# B&R Automation Studio project FASTorySystems (part 6)

#### Types.typ - Exported data types
```iecst
TYPE
	fdMove6DParametersType : 	STRUCT
		Position : fdMove6DParPositionType;
		Limits : fdMove6DParLimitsType;
		Velocity : fdMove6DParVelocityType;
		Mode : McAcp6DMoveModeEnum;
	END_STRUCT;
	fdMove6DParPositionType : 	STRUCT
		X : REAL;
		Y : REAL;
		Z : REAL;
		Rx : REAL;
		Ry : REAL;
		Rz : REAL;
	END_STRUCT;
	fdMove6DParLimitsType : 	STRUCT
		Velocity_InPlane : REAL;
		Velocity_Rx : REAL;
		Velocity_Ry : REAL;
		Velocity_Rz : REAL;
		Velocity_Z : REAL;
		Acceleration : REAL;
	END_STRUCT;
	fdMove6DParVelocityType : 	STRUCT
		InPlane : REAL;
		Z : REAL;
		Rx : REAL;
		Ry : REAL;
		Rz : REAL;
	END_STRUCT;
END_TYPE
```

#### Constants.var - Exported constants
```iecst
VAR CONSTANT
	fdMAX_STATION_SHUTTLE_COUNT : DINT := 4;
END_VAR
```

#### FastLib.fun - Exported functions and function blocks
```iecst
FUNCTION_BLOCK fdStationQueueControl
	VAR_INPUT
		Enable : {REDUND_UNREPLICABLE} BOOL;
		ReleaseShuttles : {REDUND_UNREPLICABLE} BOOL;
		SelectNextShuttle : {REDUND_UNREPLICABLE} BOOL;
		ShuttleList : {REDUND_UNREPLICABLE} ARRAY[0..fdMAX_STATION_SHUTTLE_COUNT] OF MpTrafficShuttleInfoType;
		ShuttleCapacity : {REDUND_UNREPLICABLE} DINT; (*Count how many shuttles process station can handle*)
		pStationControl : REFERENCE TO MpTrafficStationControl;
	END_VAR
	VAR_OUTPUT
		ShuttleReleaseDone : BOOL;
		ShuttleReleaseError : BOOL;
		ReleaseShuttle : BOOL;
		LastReleasedShuttleID : UINT;
	END_VAR
	VAR
		state : DINT;
		i : DINT;
		index : DINT;
		shuttleID : UINT;
		lastSelectedIndex : UINT;
	END_VAR
END_FUNCTION_BLOCK

FUNCTION_BLOCK fdTiltAround
	VAR_INPUT
		Execute : {REDUND_UNREPLICABLE} BOOL;
		MaxAngle : {REDUND_UNREPLICABLE} REAL;
		Steps : {REDUND_UNREPLICABLE} DINT;
		Velocity : McAcp6DShortAxAxesType;
		Shuttle : REFERENCE TO Mc6DShuttleType;
	END_VAR
	VAR_OUTPUT
		Acknowledge : BOOL;
		Error : BOOL;
	END_VAR
	VAR
		state : DINT;
		step : DINT;
		MoveShortAxis : MC_BR_MoveShortAxis_Acp6D;
	END_VAR
END_FUNCTION_BLOCK

FUNCTION_BLOCK fdWaitUntilAllDone
	VAR_INPUT
		Execute : {REDUND_UNREPLICABLE} BOOL;
		Shuttles : {REDUND_UNREPLICABLE} ARRAY[0..fdMAX_STATION_SHUTTLE_COUNT] OF Mc6DShuttleType;
	END_VAR
	VAR_OUTPUT
		Done : BOOL;
		Error : BOOL;
		WaitingFor : UINT;
	END_VAR
	VAR
		state : DINT;
		i : DINT;
		ShGetInfo : MC_BR_ShGetInfo_Acp6D;
	END_VAR
END_FUNCTION_BLOCK

FUNCTION_BLOCK fdPulse
	VAR_INPUT
		Execute : {REDUND_UNREPLICABLE} BOOL;
		T_on : {REDUND_UNREPLICABLE} TIME;
		T_off : {REDUND_UNREPLICABLE} TIME;
	END_VAR
	VAR_OUTPUT
		Q : BOOL;
	END_VAR
	VAR
		state : DINT;
		TON_on : TON;
		TON_off : TON;
	END_VAR
END_FUNCTION_BLOCK

FUNCTION_BLOCK fdLampSequence
	VAR_INPUT
		Execute : {REDUND_UNREPLICABLE} BOOL;
	END_VAR
	VAR_OUTPUT
		Lamp1 : BOOL;
		Lamp2 : BOOL;
		Lamp3 : BOOL;
	END_VAR
	VAR
		state : DINT;
		TON_delay : TON;
	END_VAR
END_FUNCTION_BLOCK

FUNCTION_BLOCK fdFindZone
	VAR_INPUT
		Assembly : REFERENCE TO Mc6DAssemblyType; (*The assembly reference establishes the connection between the function block and the assembly.*)
		Execute : BOOL;
		Name : STRING[32];
	END_VAR
	VAR_OUTPUT
		ZoneFound : BOOL;
		ZoneNotFound : BOOL;
		Error : BOOL;
		Zone : Mc6DZoneType; (* Zone reference *)
		ZoneInfo : McAcp6DGetZoneAddInfoType;
	END_VAR
	VAR
		state : DINT;
		i : DINT;
		AsmGetZone : MC_BR_AsmGetZone_Acp6D;
		lastZoneID : UINT;
	END_VAR
END_FUNCTION_BLOCK

FUNCTION_BLOCK fdMove6D
	VAR_INPUT
		Shuttle : REFERENCE TO Mc6DShuttleType; (*The assembly reference establishes the connection between the function block and the assembly.*)
		Execute : BOOL;
		Parameters : fdMove6DParametersType;
	END_VAR
	VAR_OUTPUT
		Acknowledge : BOOL;
		Done : BOOL;
		Error : BOOL;
	END_VAR
	VAR
		state : DINT;
		i : DINT;
		ShGetInfo : MC_BR_ShGetInfo_Acp6D;
		Move6D : MC_BR_Move6D_Acp6D;
	END_VAR
END_FUNCTION_BLOCK
```

#### fdReleaseQueuingShuttle.st
```iecst
(*  *)
FUNCTION_BLOCK fdStationQueueControl

	IF NOT Enable THEN
		state := 0;
		ReleaseShuttle := FALSE;
		SelectNextShuttle := FALSE;
		LastReleasedShuttleID := 0;
		ShuttleReleaseDone := FALSE;
		ShuttleReleaseError := FALSE;
		RETURN;
	END_IF;

	CASE state OF
		0:
			// -----------------------------------------------------------------
			SelectNextShuttle := FALSE;

			IF ReleaseShuttles THEN
				state := 20;
			ELSIF pStationControl.Info.NumOccupyingShuttles > ShuttleCapacity THEN
				// Station is executing current process and there is no room for more shuttles ->
				// release queuing extra shuttles straight forward
				state := 10;
			END_IF;
		10:
			// Check if we have our last arrived shuttle selected
			// -----------------------------------------------------------------
			IF pStationControl.SelectedShuttle.ShuttleID = pStationControl.Info.LastArrivedShuttle.ShuttleID THEN
	  			state := 12;
			ELSE
				lastSelectedIndex := pStationControl.SelectedShuttle.Index;
				SelectNextShuttle := FALSE;
				state := 11;
			END_IF;
		11:
			// Select next shuttle in the queue
			// -----------------------------------------------------------------
			SelectNextShuttle := TRUE;
			// Wait until selection changes
			IF lastSelectedIndex <> pStationControl.SelectedShuttle.Index THEN
				SelectNextShuttle := FALSE;
				state := 10;
			END_IF;
		12:
			// Release the queuing shuttle
			// -----------------------------------------------------------------
			ReleaseShuttle := TRUE;

			IF pStationControl.ReleaseDone THEN
				LastReleasedShuttleID := pStationControl.SelectedShuttle.ShuttleID;
				ReleaseShuttle := FALSE;
				state := 0;
			ELSIF pStationControl.ReleaseAborted THEN
				LastReleasedShuttleID := 0;
				ReleaseShuttle := FALSE;
				state := 0;
			END_IF;

		20:
			// Initialize for realease
			// -----------------------------------------------------------------
			i := 0;
			state := 21;
		21:
			// Select the next requested shuttle from the shuttle list
			// -----------------------------------------------------------------
			shuttleID := 0;

			WHILE i <= fdMAX_STATION_SHUTTLE_COUNT DO
				IF ShuttleList[i].ShuttleID > 0 THEN
					shuttleID := ShuttleList[i].ShuttleID;
					i := i + 1;
					EXIT;
				END_IF;
				i := i + 1;
			END_WHILE;

			IF shuttleID > 0 THEN
				// Found shuttle to release
				state := 22;
			ELSE
				// No more shuttles to release
	  			state := 100;
			END_IF;
		22:
			// Check if we have our last arrived shuttle selected
			// -----------------------------------------------------------------
			IF pStationControl.SelectedShuttle.ShuttleID = shuttleID THEN
				state := 24;
			ELSE
				lastSelectedIndex := pStationControl.SelectedShuttle.Index;
				SelectNextShuttle := FALSE;
				state := 23;
			END_IF;
		23:
			// Select next shuttle in the queue
			// -----------------------------------------------------------------
			SelectNextShuttle := TRUE;
			// Wait until selection changes
			IF lastSelectedIndex <> pStationControl.SelectedShuttle.Index THEN
				SelectNextShuttle := FALSE;
				i := 0;
				state := 21;
			END_IF;
		24:
			// Release the queuing shuttle
			// -----------------------------------------------------------------
			ReleaseShuttle := TRUE;

			IF pStationControl.ReleaseDone THEN
				LastReleasedShuttleID := pStationControl.SelectedShuttle.ShuttleID;
				ReleaseShuttle := FALSE;
				state := 21;
			ELSIF pStationControl.ReleaseAborted THEN
				LastReleasedShuttleID := 0;
				ReleaseShuttle := FALSE;
				state := 21;
			END_IF;

//
//		22:
//			// Find shuttle from stations shuttle table
//			// -----------------------------------------------------------------
//			state := 21; // Assume we dont find shuttle and just return straight to next one
//
//			FOR index := 0 TO pStationControl.Info.NumOccupyingShuttles DO
//				IF pStationControl.SelectedShuttle.ShuttleID = shuttleID THEN
//					state := 23;
//					EXIT;
//				END_IF
//				pStationControl(SelectNextShuttle := TRUE);
//				pStationControl(SelectNextShuttle := FALSE);
//			END_FOR;
//
//		23:
//			// Release the waiting shuttle
//			// -----------------------------------------------------------------
//			ReleaseShuttle := TRUE;
//
//			IF pStationControl.ReleaseDone THEN
//				ReleaseShuttle := FALSE;
//				state := 21;
//			END_IF;
		100:
			// Done
			// -----------------------------------------------------------------
			IF NOT ReleaseShuttles THEN
				state := 0;
			END_IF;
		200:
			// Error
			// -----------------------------------------------------------------
			IF NOT ReleaseShuttles THEN
				state := 0;
			END_IF;
	END_CASE;

	ShuttleReleaseDone := (state = 100);
	ShuttleReleaseError := (state = 200);

END_FUNCTION_BLOCK
```

#### fdTiltAround.st
```iecst
(*  *)
FUNCTION_BLOCK fdTiltAround

	IF NOT Execute THEN
		MoveShortAxis.Execute := FALSE;
		step := 0;
		state := 0;
	END_IF;

	CASE state OF
		0:
			IF Execute THEN
				state := 10;
			END_IF;
		10:
			IF step > Steps THEN
				state := 100;
			ELSE
				MoveShortAxis.Parameters.Position.Rx := MaxAngle * SIN((2 * brmPI / Steps) * step);
				MoveShortAxis.Parameters.Position.Ry := MaxAngle * COS((2 * brmPI / Steps) * step);
				MoveShortAxis.Parameters.Position.Rz := 0;
				MoveShortAxis.Parameters.Position.Z := 0.004;
				state := 20;
			END_IF;
		20:
			MoveShortAxis.Execute := TRUE;

			IF MoveShortAxis.Acknowledge THEN
				MoveShortAxis.Execute := FALSE;
				step := step + 1;
				state := 10;
			END_IF;
		100:
//			MoveShortAxis.Parameters.Position.Rx := 0;
//			MoveShortAxis.Parameters.Position.Ry := 0;
//			MoveShortAxis.Parameters.Position.Rz := 0;
//			MoveShortAxis.Parameters.Position.Z := 0.001;
//			MoveShortAxis.Execute := TRUE;
//
//			IF MoveShortAxis.Done OR MoveShortAxis.Acknowledge THEN
//				MoveShortAxis.Execute := FALSE;
//				step := step + 1;
//				state := 101;
//			END_IF;

			IF NOT Execute THEN
				state := 0;
			END_IF;
	END_CASE;

	MoveShortAxis.Shuttle := ADR(Shuttle);
	MoveShortAxis.Parameters.Mode :=  mcACP6D_MOVE_ABSOLUTE;
	MoveShortAxis.Parameters.Velocity := Velocity;
	MoveShortAxis();

	Acknowledge := (state = 100);
	Error := MoveShortAxis.Error;

END_FUNCTION_BLOCK
```

#### fdWaitUntilIdle.st
```iecst
(*  *)
FUNCTION_BLOCK fdWaitUntilAllDone

	IF NOT Execute THEN
		state := 0;
		i := 0;
		ShGetInfo.Execute := FALSE;
		WaitingFor := 0;
	END_IF;

	CASE state OF
		0:
			IF Execute THEN
				state := 10;
			END_IF;
		10:
			IF i > fdMAX_STATION_SHUTTLE_COUNT THEN
				state := 100;
			ELSE
				IF Shuttles[i].controlif = 0 THEN
					// Not a valid shuttle reference. Move to next item in the list
					i := i + 1;
				ELSE
					state := 20;
				END_IF;
			END_IF;
		20:
			ShGetInfo.Execute := TRUE;

			IF ShGetInfo.Done THEN
				WaitingFor := ShGetInfo.ShuttleInfo.ShuttleID;

				IF (ShGetInfo.ShuttleInfo.State =  mcACP6D_SH_STATE_IDLING) AND (ShGetInfo.ShuttleInfo.MotionBuffer.NumberOfCommands = 0) THEN
					i := i + 1;
					state := 10;
				END_IF;
				ShGetInfo.Execute := FALSE;

			ELSIF ShGetInfo.Error THEN
				ShGetInfo.Execute := FALSE;
				state := 101;
			END_IF;
		100:
			IF NOT Execute THEN
				state := 0;
			END_IF;
	END_CASE;

	ShGetInfo.Shuttle := ADR(Shuttles[i]);
	ShGetInfo();

	Done := (state = 100);
	Error := ShGetInfo.Error;

END_FUNCTION_BLOCK
```

#### fdPulse.st
```iecst
(*  *)
FUNCTION_BLOCK fdPulse

	IF NOT Execute THEN
		state := 0;
	END_IF;

	CASE state OF
		0:
			IF Execute THEN
				state := 10;
			END_IF;
		10:
			IF TON_on.Q THEN
	  			state := 20;
			END_IF;
		20:
			IF TON_off.Q THEN
				state := 10;
			END_IF;
		100:
			IF NOT Execute THEN
				state := 0;
			END_IF;
	END_CASE;

	TON_on.IN := (state = 10);
	TON_on.PT := T_on;
	TON_on();

	TON_off.IN := (state = 20);
	TON_off.PT := T_off;
	TON_off();

	Q := (state = 10);

END_FUNCTION_BLOCK
```

#### fdLampSequence.st
```iecst
(*  *)
FUNCTION_BLOCK fdLampSequence

	IF NOT Execute THEN
		state := 0;
	END_IF;

	CASE state OF
		0:
			IF Execute THEN
				state := 10;
			END_IF;
		10:
			TON_delay.IN := TRUE;
			IF TON_delay.Q THEN
				TON_delay.IN := FALSE;
	  			state := 20;
			END_IF;
		20:
			TON_delay.IN := TRUE;
			IF TON_delay.Q THEN
				TON_delay.IN := FALSE;
				state := 30;
			END_IF;
		30:
			TON_delay.IN := TRUE;
			IF TON_delay.Q THEN
				TON_delay.IN := FALSE;
				state := 10;
			END_IF;
	END_CASE;

	TON_delay.PT := T#150ms;
	TON_delay();

	Lamp1 := (state = 10);
	Lamp2 := (state = 20);
	Lamp3 := (state = 30);

END_FUNCTION_BLOCK
```

#### fdFindZone.st
```iecst
(*  *)
FUNCTION_BLOCK fdFindZone

	IF NOT Execute THEN
		state := 0;
		i := 0;
		AsmGetZone.Enable := FALSE;
		ZoneFound := FALSE;
		ZoneNotFound := FALSE;
		Error := FALSE;
		brsmemset(ADR(ZoneInfo), 0, SIZEOF(ZoneInfo));
		brsmemset(ADR(Zone), 0, SIZEOF(Zone));
	END_IF;

	CASE state OF
		0:
			// --------------------------------------------
			IF Execute THEN
				state := 10;
			END_IF;
		10:
			// --------------------------------------------
			AsmGetZone.Enable := TRUE;
			IF AsmGetZone.Valid THEN
				IF AsmGetZone.TotalCount = 0 THEN
					state := 101;
				ELSE
					state := 20;
				END_IF;
			END_IF;
		20:
			// --------------------------------------------
			lastZoneID := AsmGetZone.AdditionalInfo.ZoneID;

			IF brsmemcmp(ADR(AsmGetZone.AdditionalInfo.Name), ADR(Name), SIZEOF(Name)) = 0 THEN
				// Names match -> found
				Zone := AsmGetZone.Zone;
				ZoneInfo := AsmGetZone.AdditionalInfo;
				state := 100;
			ELSE
				IF AsmGetZone.RemainingCount = 0 THEN
					state := 101;
				ELSE
					state := 30;
				END_IF;
			END_IF;
		30:
			// --------------------------------------------
			IF AsmGetZone.AdditionalInfo.ZoneID <> lastZoneID THEN
				state := 20;
			END_IF;

		100:
			// --------------------------------------------
			ZoneFound := TRUE;
		101:
			// --------------------------------------------
			ZoneNotFound := TRUE;
		102:
			// --------------------------------------------
			Error := TRUE;
	END_CASE;

	AsmGetZone.Assembly := ADR(Assembly);
	AsmGetZone.Next := (state = 30);
	AsmGetZone();

END_FUNCTION_BLOCK
```

#### fdMove6D.st
```iecst
(*  *)
FUNCTION_BLOCK fdMove6D

//	IF NOT Execute THEN
//		state := 0;
//		i := 0;
//	END_IF;
//
//	CASE state OF
//		0:
//			// --------------------------------------------
//			IF Execute THEN
//				state := 10;
//			END_IF;
//		100:
//			// --------------------------------------------
//			ZoneFound := TRUE;
//		101:
//			// --------------------------------------------
//			ZoneNotFound := TRUE;
//		102:
//			// --------------------------------------------
//			Error := TRUE;
//	END_CASE;
//
//	Move6D.Assembly := ADR(Shuttle);
//	AsmGetZone.Next := (state = 30);
//	AsmGetZone();
//
//	ShGetInfo.Shuttle := ADR(Shuttle);
//	ShGetInfo();

END_FUNCTION_BLOCK
```

### global.var
```iecst
VAR
	gFastDemo : FastDemoType := (0);
END_VAR
```

### global.typ
```iecst
(*
Program: FastDemo

Description
(short summary)

*)
(*========== INPUTS ==========*)

TYPE
	FastDemoInputCommandType : 	STRUCT
		Activate : BOOL;
	END_STRUCT;
	FastDemoInputStatusType : 	STRUCT
		SetupComplete : BOOL;
	END_STRUCT;
	FastDemoInputType : 	STRUCT
		Force : BOOL;
		Command : FastDemoInputCommandType;
		Status : FastDemoInputStatusType;
	END_STRUCT;
END_TYPE

(*========== OUTPUTS ==========*)

TYPE
	FastDemoOutputCommandType : 	STRUCT
		NewCommand : BOOL;
	END_STRUCT;
	FastDemoOutputStatusType : 	STRUCT
		NewStatus : BOOL;
	END_STRUCT;
	FastDemoOutputType : 	STRUCT
		Command : FastDemoOutputCommandType;
		Status : FastDemoOutputStatusType;
	END_STRUCT;
END_TYPE

(*========== ERRORS ==========*)
(*========== SETTINGS ==========*)

TYPE
	FastDemoSettingsType : 	STRUCT
		Enable : BOOL;
	END_STRUCT;
END_TYPE

(*========== INTERFACE ==========*)

TYPE
	FastDemoType : 	STRUCT
		Error : GeneralErrorInfoType;
		Input : FastDemoInputType;
		Output : FastDemoOutputType;
		Settings : FastDemoSettingsType;
	END_STRUCT;
END_TYPE
```

### Program Logical/src/FastDemo/FastDemo (IEC)

#### FastDemo.st
```iecst
PROGRAM _INIT

    // Access the task interface
    task ACCESS ADR(gFastDemo);

    // Register module config interface for common setup/parametrization functionality
    //fb.MpRecipeRegPar_settings(MpLink := ADR(gSystemSettings), Enable := TRUE , PVName := ADR('gFastDemo.settings'), Category := ADR('FastDemo'));

    // Check for simulator
    //task.IsSimulated := DiagCpuIsSimulated();

    // PackML setup
    // =================================================================================================================
    em.Setup.Name := 'FastDemo';
	em.Setup.ParentName := 'Main';

END_PROGRAM

PROGRAM _CYCLIC

    // Access task interface
    // =================================================================================================================
    task ACCESS ADR(gFastDemo);

    // Inputs
    // =================================================================================================================
    IF NOT task.Input.Force THEN

    END_IF

	// Task state machine
	// =================================================================================================================
	// PackML state machine execution
	PackML_state_machine;

	// Detect state change events
	// =================================================================================================================
	// Record information which state caused abort
	fb.R_TRIG_Abort(CLK := em.Command.Abort);

	IF fb.R_TRIG_Abort.Q THEN
		task.Error.State := em.StateCurrent;
		task.Error.SubState := em.SubState;
		task.Error.Description := em.StateInfo;
	END_IF;

	// State change event
	fb.rtStateComplete(CLK := em.Command.StateComplete);

	IF fb.rtStateComplete.Q THEN
		em.StateInfo := '';
		brsmemset(ADR(actions_state), 0, SIZEOF(actions_state));

		// Record information which state caused abort
		IF em.StateCurrent = STATE_ABORTING THEN
			task.Error.State := local.lastState;
			task.Error.SubState := local.lastSubState;
			task.Error.Description := local.lastStateInfo;
		END_IF;

		FOR station_num := 0 TO STATION_COUNT DO
			// Reset station commands when major state changes
			stations[station_num].State := 0;
			brsmemset(ADR(stations[station_num].Var), 0, SIZEOF(stations[station_num].Var));
			brsmemset(ADR(stations[station_num].Commands), 0, SIZEOF(stations[station_num].Commands));
			stations[station_num].Macro.Execute := FALSE;
		END_FOR;
	END_IF;

	// Substate changed event
	IF em.SubState <> local.lastSubState THEN
		em.StateInfo := '';
		brsmemset(ADR(actions_substate), 0, SIZEOF(actions_substate));
		local.lastSubState := em.SubState;
	END_IF;

	// PackML equipment module
	// =================================================================================================================
	em();

	// Function calls
    // =================================================================================================================
	fb.TrafficControl.Enable := TRUE;
	fb.TrafficControl.MpLink := ADR(TrafficManager_x6d_1);
	fb.TrafficControl.ActivateRecipe := actions_substate.traffic_activate_recipe;
	fb.TrafficControl.DeactivateRecipe := actions_substate.traffic_deactivate_recipe;
	fb.TrafficControl.ErrorReset := actions_state.error_reset;
	fb.TrafficControl.Halt := actions_substate.traffic_halt;
	fb.TrafficControl.Recover := actions_substate.traffic_recover;
	fb.TrafficControl.Resume := actions_substate.traffic_resume;
	fb.TrafficControl.Stop := actions_substate.traffic_stop;
	fb.TrafficControl();

	fb.TON_RecoverTimeout.IN := fb.TrafficControl.RecoverBuffered;
	fb.TON_RecoverTimeout.PT := T#5s;
	fb.TON_RecoverTimeout();

	fb.TrafficMonitor.Enable := TRUE;
	fb.TrafficMonitor.MpLink := ADR(TrafficManager_x6d_1);
	fb.TrafficMonitor();

	fb.MacroDelete.Assembly := ADR(gAssembly6D_Big);
	fb.MacroDelete.Execute := actions_substate.macro_delete;
	fb.MacroDelete.Command := mcACP6D_MACRO_DELETE_ALL;
	fb.MacroDelete();

	fb.GroupGet.Assembly := ADR(gAssembly6D_Big);
	fb.GroupGet.Enable := actions_state.group_get_enable;
	fb.GroupGet();

	fb.GroupDelete.Execute := actions_substate.group_delete;
	fb.GroupDelete();

	// Perform all common station operations
	FOR station_num := 0 TO STATION_COUNT DO
		station ACCESS ADR(stations[station_num]);

		// Station control
		station.Control.MpLink := ADR(TrafficManager_x6d_1);
		station.Control.ErrorReset := actions_state.error_reset;
		station.Control.Release := station.Operation.StationQueueControl.ReleaseShuttle;
		station.Control.SelectNextShuttle := station.Operation.StationQueueControl.SelectNextShuttle;
		station.Control();

		station.Operation.StationQueueControl.Enable := actions_state.activate_queue_control;
		station.Operation.StationQueueControl.ReleaseShuttles := station.Commands.Release;
		station.Operation.StationQueueControl.pStationControl := ADR(station.Control);
		station.Operation.StationQueueControl();

		// Movement
		station.Operation.MoveInPlane.Execute := station.Commands.MoveInPlane;
		station.Operation.MoveInPlane();

		station.Operation.MoveArc.Execute := station.Commands.MoveArc;
		station.Operation.MoveArc();

		station.Operation.Move6D.Execute := station.Commands.Move6D;
		station.Operation.Move6D();

		station.Operation.MoveShortAxis.Execute := station.Commands.MoveShortAxis;
		station.Operation.MoveShortAxis();

		station.Operation.Spin.Execute := station.Commands.Spin;
		station.Operation.Spin();

		station.Operation.TiltAround.Execute := station.Commands.TiltAround;
		station.Operation.TiltAround();

		station.Operation.SunPlanet.Execute := station.Commands.ChangePlanet;
		station.Operation.SunPlanet();

		station.Operation.GetShuttleInfo.Execute := station.Commands.GetShuttleInfo;
		station.Operation.GetShuttleInfo();

		// Macro
		station.Macro.MacroCreate.Assembly := ADR(gAssembly6D_Big);
		station.Macro.MacroCreate.Parameters.Name := station.Macro.Name;
		station.Macro.MacroCreate.Execute := station.Commands.Macro.Create;
		station.Macro.MacroCreate();

		station.Macro.MacroSave.Shuttle := ADR(station.Macro.Shuttle);
		station.Macro.MacroSave.Execute := station.Commands.Macro.Save;
		station.Macro.MacroSave();

		station.Macro.MacroRun.Name := station.Macro.Name;
		station.Macro.MacroRun.Execute := station.Macro.Execute;
		station.Macro.MacroRun();

		// Group
		station.Group.GroupCreate.Execute := station.Commands.Group.Create;
		station.Group.GroupCreate.Assembly := ADR(gAssembly6D_Big);
		station.Group.GroupCreate();

		station.Group.GroupClear.Execute := station.Commands.Group.Clear;
		station.Group.GroupClear.ShuttleGroup := ADR(station.Group.ShuttleGroup);
		station.Group.GroupClear();

		station.Group.GroupAddShuttle.Execute := station.Commands.Group.AddShuttle;
		station.Group.GroupAddShuttle.ShuttleGroup := ADR(station.Group.ShuttleGroup);
		station.Group.GroupAddShuttle();

		station.Group.GroupCoupleCtrl.Execute := station.Commands.Group.ChangeCoupling;
		station.Group.GroupCoupleCtrl.ShuttleGroup := ADR(station.Group.ShuttleGroup);
		station.Group.GroupCoupleCtrl();

		// Zone
		station.Zone.ZoneCreate.Execute := station.Commands.Zone.Create;
		station.Zone.ZoneCreate.Assembly := ADR(gAssembly6D_Big);
		station.Zone.ZoneCreate();

		station.Zone.ZoneGetBarrierInfo.Execute := station.Commands.Zone.GetBarrierInfo;
		station.Zone.ZoneGetBarrierInfo.Zone := ADR(station.Zone.Zone);
		station.Zone.ZoneGetBarrierInfo();

		station.Zone.FindZone.Execute := station.Commands.Zone.Find;
		station.Zone.FindZone.Assembly := ADR(gAssembly6D_Big);
		station.Zone.FindZone();

		// Virtual
		station.Virtual.VirtualShCreate.Execute := station.Commands.CreateVirtualShuttle;
		station.Virtual.VirtualShCreate.Assembly := ADR(gAssembly6D_Big);
		station.Virtual.VirtualShCreate();

		// Wait
		station.Operation.WaitCommandLabel.Execute := station.Commands.WaitCommandLabel;
		station.Operation.WaitCommandLabel();

		station.Operation.WaitUntilAllDone.Execute := station.Commands.WaitUntilAllDone;
		station.Operation.WaitUntilAllDone();
	END_FOR;

	// Task outputs
	// =================================================================================================================

	// Task diagnostics
	// =================================================================================================================
	gTasks.FastDemo.State := em.StateCurrent;
	gTasks.FastDemo.SubState := em.SubState;
	gTasks.FastDemo.Mode := em.ModeID;
	gTasks.FastDemo.StateComplete := em.Command.StateComplete;
	gTasks.FastDemo.StateInfo := em.StateInfo;
	gTasks.FastDemo.WaitingForTask := em.Info.WaitingFor.Name;
	gTasks.FastDemo.Error := task.Error;

END_PROGRAM

PROGRAM _EXIT

END_PROGRAM
```

#### local.typ
```iecst
TYPE
	FastDemoFbType : 	STRUCT
		MpRecipeRegPar_settings : BOOL;
		TrafficControl : MpTrafficControl;
		TrafficMonitor : MpTrafficMonitor;
		rtStateComplete : R_TRIG;
		MacroDelete : MC_BR_MacroDelete_Acp6D;
		GroupGet : MC_BR_AsmGetShGroup_Acp6D;
		GroupDelete : MC_BR_ShGroupDelete_Acp6D;
		R_TRIG_Abort : R_TRIG;
		TON_RecoverTimeout : TON;
	END_STRUCT;
	FastDemoLocalType : 	STRUCT
		lastState : DINT;
		lastSubState : DINT;
		lastStateInfo : STRING[80];
		allGroupsDeleted : BOOL;
	END_STRUCT;
	FastDemoActionsStateType : 	STRUCT
		error_reset : BOOL;
		group_get_enable : BOOL;
		activate_queue_control : BOOL;
	END_STRUCT;
	FastDemoActionsSubstateType : 	STRUCT
		traffic_activate_recipe : BOOL; (*Task actions are not automatically reset*)
		traffic_deactivate_recipe : BOOL; (*Task actions are not automatically reset*)
		traffic_halt : BOOL;
		traffic_recover : BOOL;
		traffic_resume : BOOL;
		traffic_stop : BOOL;
		macro_delete : BOOL;
		group_delete : BOOL;
	END_STRUCT;
	FastDemoHmiType : 	STRUCT
		isRunning : BOOL;
	END_STRUCT;
END_TYPE

(**)
(*Stations*)

TYPE
	FastDemoStationType : 	STRUCT
		State : DINT;
		SequenceStep : DINT;
		Shuttles : ARRAY[0..STATION_SHUTTLE_LAST_INDEX]OF MpTrafficShuttleInfoType;
		ShuttleCount : DINT;
		Var : FastDemoStationVarType;
		Control : MpTrafficStationControl;
		Commands : FastDemoStationCommandsType;
		Operation : FastDemoStationOperationType;
		Macro : FastDemoStationMacroType;
		Group : FastDemoStationGroupType;
		Zone : FastDemoStationZoneType;
		Virtual : FastDemoStationVirtualType;
	END_STRUCT;
	FastDemoStationVarType : 	STRUCT
		PreviousState : DINT;
		StateInfo : STRING[80];
		LoopNum : DINT;
	END_STRUCT;
	FastDemoStationCommandsType : 	STRUCT
		Release : BOOL;
		Macro : FastDemoStationMacroCommandsType;
		Group : FastDemoStationGroupCommandsType;
		Zone : FastDemoStationZoneCommandsType;
		CreateVirtualShuttle : BOOL;
		MoveInPlane : BOOL;
		MoveArc : BOOL;
		MoveShortAxis : BOOL;
		Move6D : BOOL;
		Spin : BOOL;
		TiltAround : BOOL;
		ChangePlanet : BOOL;
		WaitCommandLabel : BOOL;
		GetShuttleInfo : BOOL;
		WaitUntilAllDone : BOOL;
	END_STRUCT;
	FastDemoStationMacroCommandsType : 	STRUCT
		Create : BOOL;
		Save : BOOL;
		Delete : BOOL;
	END_STRUCT;
	FastDemoStationGroupCommandsType : 	STRUCT
		Create : BOOL;
		Clear : BOOL;
		Delete : BOOL;
		AddShuttle : BOOL;
		ChangeCoupling : BOOL;
	END_STRUCT;
	FastDemoStationZoneCommandsType : 	STRUCT
		Create : BOOL;
		Find : BOOL;
		GetBarrierInfo : BOOL;
	END_STRUCT;
	FastDemoStationOperationType : 	STRUCT
		StationQueueControl : fdStationQueueControl;
		MoveInPlane : MC_BR_MoveInPlane_Acp6D;
		MoveArc : MC_BR_MoveArc_Acp6D;
		Spin : MC_BR_RotaryMotionSpin_Acp6D;
		Move6D : MC_BR_Move6D_Acp6D;
		MoveShortAxis : MC_BR_MoveShortAxis_Acp6D;
		TiltAround : fdTiltAround;
		SunPlanet : MC_BR_ShPlanet_Acp6D;
		WaitCommandLabel : MC_BR_ShWaitCmdLb_Acp6D;
		GetShuttleInfo : MC_BR_ShGetInfo_Acp6D;
		WaitUntilAllDone : fdWaitUntilAllDone;
	END_STRUCT;
	FastDemoStationMacroType : 	STRUCT
		Shuttle : Mc6DShuttleType;
		Name : STRING[32];
		Execute : BOOL;
		MacroCreate : MC_BR_MacroCreate_Acp6D;
		MacroSave : MC_BR_MacroSave_Acp6D;
		MacroRun : MC_BR_MacroRun_Acp6D;
	END_STRUCT;
	FastDemoStationGroupType : 	STRUCT
		ShuttleGroup : Mc6DShuttleGroupType;
		GroupCreate : MC_BR_ShGroupCreate_Acp6D;
		GroupClear : MC_BR_ShGroupClear_Acp6D;
		GroupCoupleCtrl : MC_BR_ShGroupCoupleCtrl_Acp6D;
		GroupAddShuttle : MC_BR_ShGroupAddShuttle_Acp6D;
	END_STRUCT;
	FastDemoStationZoneType : 	STRUCT
		Zone : Mc6DZoneType;
		Name : STRING[32];
		ZoneCreate : MC_BR_ZoneCreate_Acp6D;
		ZoneGetBarrierInfo : MC_BR_ZoneGetBarrierInfo_Acp6D;
		FindZone : fdFindZone;
	END_STRUCT;
	FastDemoStationVirtualType : 	STRUCT
		Shuttle : Mc6DShuttleType;
		ShuttleID : UINT;
		VirtualShCreate : MC_BR_VirtualShCreate_Acp6D;
	END_STRUCT;
END_TYPE
```

#### local.var
```iecst
VAR
	task : REFERENCE TO FastDemoType;
	local : FastDemoLocalType;
	fb : FastDemoFbType;
	hmi : FastDemoHmiType;
	actions_state : FastDemoActionsStateType;
	actions_substate : FastDemoActionsSubstateType;
END_VAR
(* ----- PackML ----- *)
VAR
	em : EquipmentModule;
END_VAR
(*----- Stations ----*)
VAR
	station_num : {REDUND_UNREPLICABLE} DINT := 0;
	str : STRING[80];
	i : DINT;
END_VAR
VAR CONSTANT
	STATION_COUNT : DINT := 7;
	STATION_SHUTTLE_COUNT : DINT := 4;
	STATION_SHUTTLE_LAST_INDEX : DINT := STATION_SHUTTLE_COUNT-1;
END_VAR
VAR
	stations : ARRAY[0..STATION_COUNT] OF FastDemoStationType;
	station : REFERENCE TO FastDemoStationType;
END_VAR
```

#### PackML.st
```iecst
// PackML state machine. Split into different sections that handle
// different logical sequences of PackML stadards' steps
// INFO: Add mode specific code into states by adding CASE structure
// 	CASE em.ModeID OF
//		MODE_PRODUCTION:
//			*CODE*;
//		MODE_MAINTENANCE:
//			*CODE*;
//		MODE_MANUAL:
//			*CODE*;
//		END_CASE
// -----------------------------------------------------------------

ACTION PackML_state_machine:
	// =================================================================================================================
    // Global PackML events
    // =================================================================================================================

    // =================================================================================================================
    // Normal work sequence
    // =================================================================================================================
    CASE em.StateCurrent OF
        STATE_STOPPED:
            em.StateInfo := '';
            // -----------------------------------------------------------------
            em.Command.StateComplete := TRUE;

        STATE_RESETTING:
			CASE em.SubState OF
				0:
					em.StateInfo := 'Reset traffic control errors';
					// -----------------------------------------------------------------
					actions_state.error_reset := TRUE;
					IF NOT fb.TrafficControl.Error THEN
	  					em.SubState := 10;
					END_IF;
				10:
					em.StateInfo := 'Delete all macros';
					// -----------------------------------------------------------------
					actions_substate.macro_delete := TRUE;
					IF fb.MacroDelete.Done THEN
						FOR station_num := 0 TO STATION_COUNT DO
							brsmemset(ADR(stations[station_num].Macro.Shuttle), 0, SIZEOF(stations[station_num].Macro.Shuttle));
						END_FOR;
						em.SubState := 20;
					END_IF;
				20:
					em.StateInfo := 'Delete all groups';
					// -----------------------------------------------------------------
					actions_state.group_get_enable := TRUE;

					IF fb.GroupGet.Valid THEN
						IF fb.GroupGet.TotalCount = 0 THEN
							// Clear all shuttle group references
							FOR station_num := 0 TO STATION_COUNT DO
	  							brsmemset(ADR(stations[station_num].Group.ShuttleGroup), 0, SIZEOF(stations[station_num].Group.ShuttleGroup));
							END_FOR;
	  						em.SubState := 100;
						ELSE
							fb.GroupDelete.ShuttleGroup := ADR(fb.GroupGet.ShuttleGroup);
							actions_substate.group_delete := TRUE;
							IF fb.GroupDelete.Done THEN
								// Get next group in the assembly
								fb.GroupGet(Next := TRUE);
								fb.GroupGet(Next := FALSE);
								actions_substate.group_delete := FALSE;
							END_IF;
						END_IF;
					END_IF;
				100:
					em.StateInfo := 'Reset complete';
					// -----------------------------------------------------------------
					em.Command.StateComplete := TRUE;
			END_CASE;

		STATE_IDLE:
			em.StateInfo := '';
			// -----------------------------------------------------------------
			em.Command.StateComplete := TRUE;

		STATE_STARTING:
			CASE em.SubState OF
				0:
					em.StateInfo := 'Move shuttles to recovery points';
					// -----------------------------------------------------------------
					fb.TrafficControl.Velocity := 1.8;
					fb.TrafficControl.Acceleration := 8.0;
					actions_substate.traffic_recover := TRUE;

					IF fb.TrafficControl.RecoverDone OR fb.TON_RecoverTimeout.Q THEN
						em.SubState := 10;
					END_IF;
				10:
					em.StateInfo := 'Activating traffic recipe';
					// -----------------------------------------------------------------
					actions_substate.traffic_activate_recipe := TRUE;

					IF fb.TrafficControl.ActivateRecipeDone THEN
						em.SubState := 100;
					END_IF;
				100:
					em.StateInfo := 'Traffic manager started';
					// -----------------------------------------------------------------
					IF fb.TrafficControl.Error THEN
	  					em.SubState := 200;
					ELSE
						em.Command.StateComplete := TRUE;
					END_IF;
			END_CASE;

        STATE_EXECUTE:
            em.StateInfo := 'Running feature demo';
            // -----------------------------------------------------------------
			em.Command.StateComplete := TRUE;

			actions_state.activate_queue_control := TRUE;

			execute_station_S1;
			execute_station_S2;
			execute_station_S3;
			execute_station_S4;
			execute_station_S5;
			execute_station_S6;
			//execute_station_S7;

        STATE_COMPLETING:
            em.StateInfo := '';
            // -----------------------------------------------------------------
            em.Command.StateComplete := TRUE;

        STATE_COMPLETED:
            em.StateInfo := '';
            // -----------------------------------------------------------------
            em.Command.StateComplete := TRUE;

        STATE_STOPPING:
            em.StateInfo := 'Stop traffic manager';
			// -----------------------------------------------------------------
			actions_substate.traffic_stop := TRUE;
			IF fb.TrafficControl.StopDone THEN
	  			em.Command.StateComplete := TRUE;
			END_IF;
	END_CASE

    // =================================================================================================================
    // Module activation sequence
    // =================================================================================================================
    CASE em.StateCurrent OF
        STATE_DEACTIVATING:
            em.StateInfo := '';
            // -----------------------------------------------------------------
            em.Command.StateComplete := TRUE;

        STATE_DEACTIVATED:
            em.StateInfo := '';
            // -----------------------------------------------------------------
            em.Command.StateComplete := TRUE;

        STATE_ACTIVATING:
            em.StateInfo := '';
            // -----------------------------------------------------------------
            em.Command.StateComplete := TRUE;

    END_CASE

    // =================================================================================================================
    // Abort sequence
    // =================================================================================================================
    CASE em.StateCurrent OF
        STATE_ABORTING:
            em.StateInfo := '';
            // -----------------------------------------------------------------
            em.Command.StateComplete := TRUE;

        STATE_ABORTED:
            em.StateInfo := '';
            // -----------------------------------------------------------------
            em.Command.StateComplete := TRUE;

        STATE_CLEARING:
            em.StateInfo := '';
            // -----------------------------------------------------------------
            em.Command.StateComplete := TRUE;
    END_CASE

    // =================================================================================================================
    // Hold sequence
    // =================================================================================================================
    CASE em.StateCurrent OF
        STATE_HOLDING:
            em.StateInfo := '';
            // -----------------------------------------------------------------
            em.Command.StateComplete := TRUE;

        STATE_HELD:
            em.StateInfo := '';
            // -----------------------------------------------------------------
            em.Command.StateComplete := TRUE;

        STATE_UNHOLDING:
            em.StateInfo := '';
            // -----------------------------------------------------------------
            em.Command.StateComplete := TRUE;
    END_CASE

    // =================================================================================================================
    // Suspend sequence
    // =================================================================================================================
    CASE em.StateCurrent OF
        STATE_SUSPENDING:
            em.StateInfo := '';
            // -----------------------------------------------------------------
            em.Command.StateComplete := TRUE;

        STATE_SUSPENDED:
            em.StateInfo := '';
            // -----------------------------------------------------------------
            em.Command.StateComplete := TRUE;

        STATE_UNSUSPENDING:
            em.StateInfo := '';
            // -----------------------------------------------------------------
            em.Command.StateComplete := TRUE;

    END_CASE

END_ACTION
```

#### defaults.st
```iecst
ACTION reset_parameters_all:
	reset_parameters_MoveInPlane;
	reset_parameters_MoveShortAxis;
	reset_parameters_MoveArc;
	reset_parameters_Move6D;
END_ACTION

ACTION reset_parameters_MoveInPlane:
	brsmemset(ADR(station.Operation.MoveInPlane.Parameters), 0, SIZEOF(station.Operation.MoveInPlane.Parameters));

	station.Operation.MoveInPlane.CommandLabel := 0;
	station.Operation.MoveInPlane.Parameters.Velocity := 1.5;
	station.Operation.MoveInPlane.Parameters.Acceleration := 18;
	station.Operation.MoveInPlane.Parameters.EndVelocity := 0;
	station.Operation.MoveInPlane.Parameters.Path :=  mcACP6D_PATH_DIRECT;
	station.Operation.MoveInPlane.Parameters.Mode :=  mcACP6D_MOVE_ABSOLUTE;
END_ACTION

ACTION reset_parameters_MoveShortAxis:
	brsmemset(ADR(station.Operation.MoveShortAxis.Parameters), 0, SIZEOF(station.Operation.MoveShortAxis.Parameters));

	station.Operation.MoveShortAxis.CommandLabel := 0;
	station.Operation.MoveShortAxis.Parameters.Velocity.Rx := 0.1;
	station.Operation.MoveShortAxis.Parameters.Velocity.Ry := 0.1;
	station.Operation.MoveShortAxis.Parameters.Velocity.Rz := 0.1;
	station.Operation.MoveShortAxis.Parameters.Velocity.Z := 0.005;
	station.Operation.MoveShortAxis.Parameters.Position.Rx := 0;
	station.Operation.MoveShortAxis.Parameters.Position.Ry:= 0;
	station.Operation.MoveShortAxis.Parameters.Position.Rz := 0;
	station.Operation.MoveShortAxis.Parameters.Position.Z := gDEFAULT_Z;
	station.Operation.MoveShortAxis.Parameters.Mode := mcACP6D_MOVE_ABSOLUTE;
END_ACTION

ACTION reset_parameters_MoveArc:
	brsmemset(ADR(station.Operation.MoveArc.Parameters), 0, SIZEOF(station.Operation.MoveArc.Parameters));

	station.Operation.MoveArc.CommandLabel := 0;
	station.Operation.MoveArc.Parameters.Velocity := 1.5;
	station.Operation.MoveArc.Parameters.Acceleration := 18;
	station.Operation.MoveArc.Parameters.EndVelocity := 0;
	station.Operation.MoveArc.Parameters.Angular.Angle := 0;
	station.Operation.MoveArc.Parameters.Mode :=  mcACP6D_MOVE_RELATIVE;
	station.Operation.MoveArc.Parameters.Option := mcACP6D_ARC_ANGULAR;
END_ACTION

ACTION reset_parameters_Move6D:

END_ACTION

ACTION reset_parameters_WaitCommandLabel:
	station.Operation.WaitCommandLabel.LabelType :=  mcACP6D_SH_WAIT_CMDLB_REGULAR;
	station.Operation.WaitCommandLabel.TriggerCmdLb := 0;
	station.Operation.WaitCommandLabel.TriggerType := mcACP6D_SH_WAIT_CMDLB_START;
	station.Operation.WaitCommandLabel.TriggerXID := 0;
END_ACTION
```

#### station_S1.st
```iecst
ACTION execute_station_S1:
	// Point station reference to this station
	station ACCESS ADR(stations[1]);

	// Station control logic and mapping
	station.Control.Enable := TRUE;
	station.Control.Station := ADR(S1);
	station.Control.To := ADR(S2);
	station.Macro.Name := 'S1';
	station.Operation.StationQueueControl.ShuttleCapacity := 1;

	CASE station.State OF
		0:
			station.Var.StateInfo := 'Activating station';
			// -----------------------------------------------------------------
			IF station.Control.Active AND station.Control.State = mpTRAFFIC_ST_ON_OPEN THEN
	  			station.State := station.State + 1;
			END_IF;

		1:
			station.Var.StateInfo := 'Check if station sequence macro exists';
			// -----------------------------------------------------------------
			IF station.Macro.Shuttle.controlif > 0 THEN
				// Macro already created -> go to wait for next shuttle
				station.State := 200;
			ELSE
				station.State := station.State + 1;
			END_IF;

		2:
			station.Var.StateInfo := 'Create new macro';
			// -----------------------------------------------------------------
			station.Commands.Macro.Create := TRUE;

			IF station.Macro.MacroCreate.Done THEN
				station.Macro.Shuttle := station.Macro.MacroCreate.MacroShuttle;
	  			station.State := 10;
			END_IF;
		10:
			station.Var.StateInfo := 'Movement settings';
			// -----------------------------------------------------------------
			station.Var.LoopNum := 0;

			station.Operation.MoveInPlane.Parameters.Velocity := 2;
			station.Operation.MoveInPlane.Parameters.Acceleration := 18;
			station.Operation.MoveInPlane.Parameters.EndVelocity := 0;
			station.Operation.MoveInPlane.Parameters.Radius := 0;
			station.Operation.MoveInPlane.Parameters.Path :=  mcACP6D_PATH_DIRECT;
			station.Operation.MoveInPlane.Shuttle := ADR(station.Macro.Shuttle);

			station.State := station.State + 1;
		11:
			station.Var.StateInfo := 'Move to UL';
			// -----------------------------------------------------------------
			station.Operation.MoveInPlane.Parameters.Mode :=  mcACP6D_MOVE_ABSOLUTE;
			station.Operation.MoveInPlane.Parameters.Position.X := 0.060;
			station.Operation.MoveInPlane.Parameters.Position.Y := 0.420;
			station.Commands.MoveInPlane := TRUE;

			IF station.Operation.MoveInPlane.Acknowledge THEN
				station.State := station.State + 1;
			END_IF;
		12:
			station.Var.StateInfo := 'Move to LL';
			// -----------------------------------------------------------------
			station.Operation.MoveInPlane.Parameters.Mode :=  mcACP6D_MOVE_ABSOLUTE;
			station.Operation.MoveInPlane.Parameters.Position.X := 0.060;
			station.Operation.MoveInPlane.Parameters.Position.Y := 0.060;
			station.Commands.MoveInPlane := TRUE;

			IF station.Operation.MoveInPlane.Acknowledge THEN
				station.State := station.State + 1;
			END_IF;
		13:
			station.Var.StateInfo := 'Move to LR';
			// -----------------------------------------------------------------
			station.Operation.MoveInPlane.Parameters.Mode :=  mcACP6D_MOVE_ABSOLUTE;
			station.Operation.MoveInPlane.Parameters.Position.X := 0.180;
			station.Operation.MoveInPlane.Parameters.Position.Y := 0.060;
			station.Commands.MoveInPlane := TRUE;

			IF station.Operation.MoveInPlane.Acknowledge THEN
				station.State := station.State + 1;
			END_IF;
		14:
			station.Var.StateInfo := 'Move to UR';
			// -----------------------------------------------------------------
			station.Operation.MoveInPlane.Parameters.Mode :=  mcACP6D_MOVE_ABSOLUTE;
			station.Operation.MoveInPlane.Parameters.Position.X := 0.180;
			station.Operation.MoveInPlane.Parameters.Position.Y := 0.420;
			station.Commands.MoveInPlane := TRUE;

			IF station.Operation.MoveInPlane.Acknowledge THEN
				station.State := station.State + 1;
			END_IF;
		15:
			station.Var.StateInfo := 'Move to UL';
			// -----------------------------------------------------------------
			station.Operation.MoveInPlane.Parameters.Mode :=  mcACP6D_MOVE_ABSOLUTE;
			station.Operation.MoveInPlane.Parameters.Position.X := 0.060;
			station.Operation.MoveInPlane.Parameters.Position.Y := 0.420;
			station.Commands.MoveInPlane := TRUE;

			IF station.Operation.MoveInPlane.Acknowledge THEN
				station.State := station.State + 1;
			END_IF;
		16:
			station.Var.StateInfo := 'Move to LR';
			// -----------------------------------------------------------------
			station.Operation.MoveInPlane.Parameters.Mode :=  mcACP6D_MOVE_ABSOLUTE;
			station.Operation.MoveInPlane.Parameters.Position.X := 0.180;
			station.Operation.MoveInPlane.Parameters.Position.Y := 0.060;
			station.Commands.MoveInPlane := TRUE;

			IF station.Operation.MoveInPlane.Acknowledge THEN
				station.State := station.State + 1;
			END_IF;
		17:
			station.Var.StateInfo := 'Move to LL';
			// -----------------------------------------------------------------
			station.Operation.MoveInPlane.Parameters.Mode :=  mcACP6D_MOVE_ABSOLUTE;
			station.Operation.MoveInPlane.Parameters.Position.X := 0.060;
			station.Operation.MoveInPlane.Parameters.Position.Y := 0.060;
			station.Commands.MoveInPlane := TRUE;

			IF station.Operation.MoveInPlane.Acknowledge THEN
				station.State := station.State + 1;
			END_IF;
		18:
			station.Var.StateInfo := 'Move to UR';
			// -----------------------------------------------------------------
			station.Operation.MoveInPlane.Parameters.Mode :=  mcACP6D_MOVE_ABSOLUTE;
			station.Operation.MoveInPlane.Parameters.Position.X := 0.180;
			station.Operation.MoveInPlane.Parameters.Position.Y := 0.420;
			station.Commands.MoveInPlane := TRUE;

			IF station.Operation.MoveInPlane.Acknowledge THEN
				station.State := station.State + 1;
			END_IF;
		19:
			station.Var.StateInfo := 'Move to UL';
			// -----------------------------------------------------------------
			station.Operation.MoveInPlane.Parameters.Mode :=  mcACP6D_MOVE_ABSOLUTE;
			station.Operation.MoveInPlane.Parameters.Position.X := 0.060;
			station.Operation.MoveInPlane.Parameters.Position.Y := 0.420;
			station.Commands.MoveInPlane := TRUE;

			IF station.Operation.MoveInPlane.Acknowledge THEN
				station.State := station.State + 1;
			END_IF;
		20:
			station.Var.StateInfo := 'Move to LL';
			// -----------------------------------------------------------------
			station.Operation.MoveInPlane.Parameters.Mode :=  mcACP6D_MOVE_ABSOLUTE;
			station.Operation.MoveInPlane.Parameters.Position.X := 0.060;
			station.Operation.MoveInPlane.Parameters.Position.Y := 0.060;
			station.Commands.MoveInPlane := TRUE;

			IF station.Operation.MoveInPlane.Acknowledge THEN
				station.State := 30;
			END_IF;
		30:
			station.Var.StateInfo := 'Move right';
			// -----------------------------------------------------------------
			station.Operation.MoveInPlane.Parameters.Mode :=  mcACP6D_MOVE_RELATIVE;
			station.Operation.MoveInPlane.Parameters.Position.X := 0.120;
			station.Operation.MoveInPlane.Parameters.Position.Y := 0.000;
			station.Commands.MoveInPlane := TRUE;

			IF station.Operation.MoveInPlane.Acknowledge THEN
				station.State := station.State + 1;
			END_IF;
		31:
			station.Var.StateInfo := 'Move up';
			// -----------------------------------------------------------------
			station.Operation.MoveInPlane.Parameters.Mode :=  mcACP6D_MOVE_RELATIVE;
			station.Operation.MoveInPlane.Parameters.Position.X := 0.000;
			station.Operation.MoveInPlane.Parameters.Position.Y := 0.120;
			station.Commands.MoveInPlane := TRUE;

			IF station.Operation.MoveInPlane.Acknowledge THEN
				station.State := station.State + 1;
			END_IF;
		32:
			station.Var.StateInfo := 'Move left';
			// -----------------------------------------------------------------
			station.Operation.MoveInPlane.Parameters.Mode :=  mcACP6D_MOVE_RELATIVE;
			station.Operation.MoveInPlane.Parameters.Position.X := -0.120;
			station.Operation.MoveInPlane.Parameters.Position.Y := 0.000;
			station.Commands.MoveInPlane := TRUE;

			IF station.Operation.MoveInPlane.Acknowledge THEN
				station.State := station.State + 1;
			END_IF;
		33:
			station.Var.StateInfo := 'Move up';
			// -----------------------------------------------------------------
			station.Operation.MoveInPlane.Parameters.Mode :=  mcACP6D_MOVE_RELATIVE;
			station.Operation.MoveInPlane.Parameters.Position.X := 0.000;
			station.Operation.MoveInPlane.Parameters.Position.Y := 0.120;
			station.Commands.MoveInPlane := TRUE;

			IF station.Operation.MoveInPlane.Acknowledge THEN
				station.State := station.State + 1;
			END_IF;
		34:
			station.Var.StateInfo := 'Move right';
			// -----------------------------------------------------------------
			station.Operation.MoveInPlane.Parameters.Mode :=  mcACP6D_MOVE_RELATIVE;
			station.Operation.MoveInPlane.Parameters.Position.X := 0.120;
			station.Operation.MoveInPlane.Parameters.Position.Y := 0.000;
			station.Commands.MoveInPlane := TRUE;

			IF station.Operation.MoveInPlane.Acknowledge THEN
				station.State := station.State + 1;
			END_IF;
		35:
			station.Var.StateInfo := 'Move up';
			// -----------------------------------------------------------------
			station.Operation.MoveInPlane.Parameters.Mode :=  mcACP6D_MOVE_RELATIVE;
			station.Operation.MoveInPlane.Parameters.Position.X := 0.000;
			station.Operation.MoveInPlane.Parameters.Position.Y := 0.120;
			station.Commands.MoveInPlane := TRUE;

			IF station.Operation.MoveInPlane.Acknowledge THEN
				station.State := station.State + 1;
			END_IF;
		36:
			station.Var.StateInfo := 'Move left';
			// -----------------------------------------------------------------
			station.Operation.MoveInPlane.Parameters.Mode :=  mcACP6D_MOVE_RELATIVE;
			station.Operation.MoveInPlane.Parameters.Position.X := -0.120;
			station.Operation.MoveInPlane.Parameters.Position.Y := 0.000;
			station.Commands.MoveInPlane := TRUE;

			IF station.Operation.MoveInPlane.Acknowledge THEN
				station.State := station.State + 1;
			END_IF;
		37:
			station.Var.StateInfo := 'Move down';
			// -----------------------------------------------------------------
			station.Operation.MoveInPlane.Parameters.Mode :=  mcACP6D_MOVE_RELATIVE;
			station.Operation.MoveInPlane.Parameters.Position.X := 0.000;
			station.Operation.MoveInPlane.Parameters.Position.Y := -0.120;
			station.Commands.MoveInPlane := TRUE;

			IF station.Operation.MoveInPlane.Acknowledge THEN
				station.State := station.State + 1;
			END_IF;
		38:
			station.Var.StateInfo := 'Move right';
			// -----------------------------------------------------------------
			station.Operation.MoveInPlane.Parameters.Mode :=  mcACP6D_MOVE_RELATIVE;
			station.Operation.MoveInPlane.Parameters.Position.X := 0.120;
			station.Operation.MoveInPlane.Parameters.Position.Y := 0.000;
			station.Commands.MoveInPlane := TRUE;

			IF station.Operation.MoveInPlane.Acknowledge THEN
				station.State := station.State + 1;
			END_IF;
		39:
			station.Var.StateInfo := 'Move down';
			// -----------------------------------------------------------------
			station.Operation.MoveInPlane.Parameters.Mode :=  mcACP6D_MOVE_RELATIVE;
			station.Operation.MoveInPlane.Parameters.Position.X := 0.000;
			station.Operation.MoveInPlane.Parameters.Position.Y := -0.120;
			station.Commands.MoveInPlane := TRUE;

			IF station.Operation.MoveInPlane.Acknowledge THEN
				station.State := station.State + 1;
			END_IF;
		40:
			station.Var.StateInfo := 'Move left';
			// -----------------------------------------------------------------
			station.Operation.MoveInPlane.Parameters.Mode :=  mcACP6D_MOVE_RELATIVE;
			station.Operation.MoveInPlane.Parameters.Position.X := -0.120;
			station.Operation.MoveInPlane.Parameters.Position.Y := 0.000;
			station.Commands.MoveInPlane := TRUE;

			IF station.Operation.MoveInPlane.Acknowledge THEN
				station.State := station.State + 1;
			END_IF;
		41:
			station.Var.StateInfo := 'Move down';
			// -----------------------------------------------------------------
			station.Operation.MoveInPlane.Parameters.Mode :=  mcACP6D_MOVE_RELATIVE;
			station.Operation.MoveInPlane.Parameters.Position.X := 0.000;
			station.Operation.MoveInPlane.Parameters.Position.Y := -0.120;
			station.Commands.MoveInPlane := TRUE;

			IF station.Operation.MoveInPlane.Acknowledge THEN
				station.State := station.State + 1;
			END_IF;
		42:
			station.Var.StateInfo := 'Move right';
			// -----------------------------------------------------------------
			station.Operation.MoveInPlane.Parameters.Mode :=  mcACP6D_MOVE_RELATIVE;
			station.Operation.MoveInPlane.Parameters.Position.X := 0.120;
			station.Operation.MoveInPlane.Parameters.Position.Y := 0.000;
			station.Commands.MoveInPlane := TRUE;

			IF station.Operation.MoveInPlane.Acknowledge THEN
				station.State := 50;
			END_IF;
		50:
			station.Var.StateInfo := 'Check if sequence complete';
			// -----------------------------------------------------------------
			IF station.Var.LoopNum < 3 THEN
				station.Var.LoopNum := station.Var.LoopNum + 1;
				station.State :=  11;
			ELSE
				station.State := 100;
			END_IF;
		100:
			station.Var.StateInfo := 'Save macro';
			// -----------------------------------------------------------------
			station.Commands.Macro.Save := TRUE;

			IF station.Macro.MacroSave.Done THEN
				station.State := 200;
			END_IF;
		200:
			station.Var.StateInfo := 'Waiting for shuttle to arrive at station';
			// -----------------------------------------------------------------
			IF station.Control.Info.Occupied THEN
				station.Shuttles[0] := station.Control.Info.LastArrivedShuttle;
				station.Macro.MacroRun.Shuttle := ADR(station.Shuttles[0].Shuttle6D);
				station.State := station.State + 1;
			END_IF;
		201:
			station.Var.StateInfo := 'Wait shuttle to complete its moves';
			// -----------------------------------------------------------------
			station.Macro.Execute := TRUE;

			IF station.Macro.MacroRun.Done THEN
				station.Macro.Execute := FALSE;
				station.State := 1000;
			END_IF;
		1000:
			station.Var.StateInfo := 'Release shuttle to traffic network';
			// -----------------------------------------------------------------
			station.Operation.StationQueueControl.ShuttleList[0] := station.Shuttles[0];
			station.Commands.Release := TRUE;

			IF station.Operation.StationQueueControl.ShuttleReleaseDone THEN
				station.State := 0;
			END_IF;
	END_CASE;

	// Reset station commands when state changes
	IF station.State <> station.Var.PreviousState THEN
		station.Var.PreviousState := station.State;
		brsmemset(ADR(station.Commands), 0, SIZEOF(station.Commands));
	END_IF;

END_ACTION
```

#### station_S2.st
```iecst
ACTION execute_station_S2:
	// Point station reference to this station
	station ACCESS ADR(stations[2]);

	// Station control logic and mapping
	station.Control.Enable := TRUE;
	station.Control.Station := ADR(S2);
	station.Control.To := ADR(B1);

	CASE station.State OF
		0:
			station.Var.StateInfo := 'Activating station';
			// -----------------------------------------------------------------
			IF station.Control.Active AND station.Control.State = mpTRAFFIC_ST_ON_OPEN THEN
				station.State := station.State + 1;
			END_IF;

		1:
			station.Var.StateInfo := 'Waiting for shuttle to arrive at station';
			// -----------------------------------------------------------------
			IF station.Control.Info.Occupied THEN
				station.Operation.MoveInPlane.Shuttle := ADR(station.Control.SelectedShuttle.Shuttle6D);
				station.Operation.Spin.Shuttle := ADR(station.Control.SelectedShuttle.Shuttle6D);
	  			station.State := 10;
			END_IF;

		10:
			station.Var.StateInfo := 'Move to position 1';
			// -----------------------------------------------------------------
			station.Operation.MoveInPlane.Parameters.Velocity := 2;
			station.Operation.MoveInPlane.Parameters.Acceleration := 20;
			station.Operation.MoveInPlane.Parameters.EndVelocity := 0;

			station.Operation.MoveInPlane.Parameters.Path := mcACP6D_PATH_DIRECT;
			station.Operation.MoveInPlane.Parameters.Position.X := 0.840;
			station.Operation.MoveInPlane.Parameters.Position.Y := 0.120;

			station.Commands.MoveInPlane := TRUE;

			IF station.Operation.MoveInPlane.Acknowledge THEN
				station.State := station.State + 1;
			END_IF;

		11:
			station.Var.StateInfo := 'Spin 1';
			// -----------------------------------------------------------------
			station.Operation.Spin.Parameters.Acceleration := 35.0;
			station.Operation.Spin.Parameters.Velocity := 22.0;
			station.Operation.Spin.Parameters.Angle := 0;
			station.Operation.Spin.Parameters.Duration := 2.0;

			station.Commands.Spin := TRUE;

			IF station.Operation.Spin.Acknowledge THEN
				station.State := station.State + 1;
			END_IF;

		12:
			station.Var.StateInfo := 'Move position 2';
			// -----------------------------------------------------------------
			station.Operation.MoveInPlane.Parameters.Path := mcACP6D_PATH_DIRECT;
			station.Operation.MoveInPlane.Parameters.Position.X := 0.840;
			station.Operation.MoveInPlane.Parameters.Position.Y := 0.360;

			station.Commands.MoveInPlane := TRUE;

			IF station.Operation.MoveInPlane.Acknowledge THEN
				station.State := station.State + 1;
			END_IF;

		13:
			station.Var.StateInfo := 'Spin 2';
			// -----------------------------------------------------------------
			station.Operation.Spin.Parameters.Velocity := -22.0;

			station.Commands.Spin := TRUE;

			IF station.Operation.Spin.Done THEN
				station.State := 100;
			END_IF;

		100:
			station.Var.StateInfo := 'Check if sequence complete';
			// -----------------------------------------------------------------
			station.Var.LoopNum := station.Var.LoopNum + 1;

			IF station.Var.LoopNum > 0 THEN
				// Station sequence complete
				station.State :=  200;
			ELSE
				// New loop of moves
				station.State :=  10;
			END_IF;

		200:
			station.Var.StateInfo := 'Wait shuttle to complete its moves';
			// -----------------------------------------------------------------
			station.Operation.MoveInPlane.Parameters.Path :=  mcACP6D_PATH_DIRECT;
			station.Operation.MoveInPlane.Parameters.Position.X := 0.840;
			station.Operation.MoveInPlane.Parameters.Position.Y := 0.360;
			station.Operation.MoveInPlane.Parameters.EndVelocity := 0;

			station.Commands.MoveInPlane := TRUE;

			IF station.Operation.MoveInPlane.Done THEN
				station.State := 1000;
			END_IF;

		1000:
			station.Var.StateInfo := 'Release shuttle to traffic network';
			// -----------------------------------------------------------------
			station.Commands.Release := TRUE;

			IF station.Control.ReleaseDone THEN
				station.State := 0;
			END_IF;
	END_CASE;

	// Reset station commands when state changes
	IF station.State <> station.Var.PreviousState THEN
		station.Var.PreviousState := station.State;
		brsmemset(ADR(station.Commands), 0, SIZEOF(station.Commands));
	END_IF;

END_ACTION
```

#### station_S3.st
```iecst
ACTION execute_station_S3:
	// Point station reference to this station
	station ACCESS ADR(stations[3]);

	// Station control logic and mapping
	station.Control.Enable := TRUE;
	station.Control.Station := ADR(S3);
	station.Control.To := ADR(S5);
	station.Macro.Name := 'S3';
	station.Operation.StationQueueControl.ShuttleCapacity := 1;

	CASE station.State OF
		0:
			station.Var.StateInfo := 'Activating station';
			// -----------------------------------------------------------------
			IF station.Control.Active AND station.Control.State = mpTRAFFIC_ST_ON_OPEN THEN
				station.State := station.State + 1;
			END_IF
		1:
			station.Var.StateInfo := 'Check if station sequence macro exists';
			// -----------------------------------------------------------------
			IF station.Macro.Shuttle.controlif > 0 THEN
				// Macro already created -> go to wait for next shuttle
				station.State := 200;
			ELSE
				station.State := station.State + 1;
			END_IF
		2:
			station.Var.StateInfo := 'Create new macro';
			// -----------------------------------------------------------------
			station.Commands.Macro.Create := TRUE;

			IF station.Macro.MacroCreate.Done THEN
				station.Macro.Shuttle := station.Macro.MacroCreate.MacroShuttle;
				station.State := 10;
			END_IF;
		10:
			station.Var.StateInfo := 'Movement settings';
			// -----------------------------------------------------------------
			station.Var.LoopNum := 0;

			station.Operation.MoveInPlane.Parameters.Velocity := 2;
			station.Operation.MoveInPlane.Parameters.Acceleration := 18;
			station.Operation.MoveInPlane.Parameters.EndVelocity := 0;
			station.Operation.MoveInPlane.Parameters.Radius := 0;
			station.Operation.MoveInPlane.Parameters.Path :=  mcACP6D_PATH_DIRECT;
			station.Operation.MoveInPlane.Shuttle := ADR(station.Macro.Shuttle);

			station.Operation.MoveArc.Parameters.Acceleration := 18;
			station.Operation.MoveArc.Parameters.Velocity := 1.5;
			station.Operation.MoveArc.Parameters.EndVelocity := 1.5;
			station.Operation.MoveArc.Parameters.Mode :=  mcACP6D_MOVE_RELATIVE;
			station.Operation.MoveArc.Parameters.Option := mcACP6D_ARC_ANGULAR;
			station.Operation.MoveArc.Parameters.Angular.Angle := brmPI;
			station.Operation.MoveArc.Shuttle := ADR(station.Macro.Shuttle);

			station.State := station.State + 1;
		11:
			station.Var.StateInfo := 'Move to position 1';
			// -----------------------------------------------------------------
			station.Operation.MoveInPlane.Parameters.Position.X := 0.840;
			station.Operation.MoveInPlane.Parameters.Position.Y := 1.680;

			station.Commands.MoveInPlane := TRUE;

			IF station.Operation.MoveInPlane.Acknowledge THEN
				station.State := station.State + 1;
			END_IF;
		12:
			station.Var.StateInfo := '';
			// -----------------------------------------------------------------
			station.Operation.MoveArc.Parameters.Direction := mcACP6D_ARC_COUNTER_CLOCKWISE;
			station.Operation.MoveArc.Parameters.Angular.Center.X := 0;
			station.Operation.MoveArc.Parameters.Angular.Center.Y := 0.060;
			station.Commands.MoveArc := TRUE;

			IF station.Operation.MoveArc.Acknowledge THEN
				station.State := station.State + 1;
			END_IF;
		13:
			station.Var.StateInfo := '';
			// -----------------------------------------------------------------
			station.Operation.MoveArc.Parameters.Direction := mcACP6D_ARC_COUNTER_CLOCKWISE;
			station.Operation.MoveArc.Parameters.Angular.Center.X := 0;
			station.Operation.MoveArc.Parameters.Angular.Center.Y := -0.060;
			station.Commands.MoveArc := TRUE;

			IF station.Operation.MoveArc.Acknowledge THEN
				station.State := station.State + 1;
			END_IF;
		14:
			station.Var.StateInfo := '';
			// -----------------------------------------------------------------
			station.Operation.MoveArc.Parameters.Direction := mcACP6D_ARC_CLOCKWISE;
			station.Operation.MoveArc.Parameters.Angular.Center.X := 0;
			station.Operation.MoveArc.Parameters.Angular.Center.Y := -0.060;
			station.Commands.MoveArc := TRUE;

			IF station.Operation.MoveArc.Acknowledge THEN
				station.State := station.State + 1;
			END_IF;

		15:
			station.Var.StateInfo := '';
			// -----------------------------------------------------------------
			station.Operation.MoveArc.Parameters.Direction := mcACP6D_ARC_CLOCKWISE;
			station.Operation.MoveArc.Parameters.Angular.Center.X := 0;
			station.Operation.MoveArc.Parameters.Angular.Center.Y := 0.060;
			station.Commands.MoveArc := TRUE;

			IF station.Operation.MoveArc.Acknowledge THEN
				station.State := station.State + 1;
			END_IF;

		16:
			station.Var.StateInfo := 'Check if sequence complete';
			// -----------------------------------------------------------------
			station.Var.LoopNum := station.Var.LoopNum + 1;

			IF station.Var.LoopNum > 5 THEN
				// Station sequence complete
				station.State := station.State + 1;
			ELSE
				// New loop of moves
				station.State :=  12;
			END_IF;
		17:
			station.Var.StateInfo := 'Move to last position';
			// -----------------------------------------------------------------
			station.Operation.MoveArc.Parameters.Direction := mcACP6D_ARC_COUNTER_CLOCKWISE;
			station.Operation.MoveArc.Parameters.Angular.Center.X := 0;
			station.Operation.MoveArc.Parameters.Angular.Center.Y := 0.060;
			station.Operation.MoveArc.Parameters.EndVelocity := 0;
			station.Commands.MoveArc := TRUE;

			IF station.Operation.MoveArc.Acknowledge THEN
				station.State := 100;
			END_IF;
		100:
			station.Var.StateInfo := 'Save macro';
			// -----------------------------------------------------------------
			station.Commands.Macro.Save := TRUE;

			IF station.Macro.MacroSave.Done THEN
				station.State := 200;
			END_IF;
		200:
			station.Var.StateInfo := 'Waiting for shuttle to arrive at station';
			// -----------------------------------------------------------------
			IF station.Control.Info.Occupied THEN
				station.Shuttles[0] := station.Control.Info.LastArrivedShuttle;
				station.Macro.MacroRun.Shuttle := ADR(station.Shuttles[0].Shuttle6D);
				station.State := station.State + 1;
			END_IF;
		201:
			station.Var.StateInfo := 'Wait shuttle to complete its moves';
			// -----------------------------------------------------------------
			station.Macro.Execute := TRUE;

			IF station.Macro.MacroRun.Done THEN
				station.Macro.Execute := FALSE;
				station.State := 1000;
			END_IF;
		1000:
			station.Var.StateInfo := 'Release shuttle to traffic network';
			// -----------------------------------------------------------------
			station.Operation.StationQueueControl.ShuttleList[0] := station.Shuttles[0];
			station.Commands.Release := TRUE;

			IF station.Operation.StationQueueControl.ShuttleReleaseDone THEN
				station.State := 0;
			END_IF;
	END_CASE;

	// Reset station commands when state changes
	IF station.State <> station.Var.PreviousState THEN
		station.Var.PreviousState := station.State;
		brsmemset(ADR(station.Commands), 0, SIZEOF(station.Commands));
	END_IF;

END_ACTION
```

#### station_S4.st
```iecst
ACTION execute_station_S4:
	// Point station reference to this station
	station ACCESS ADR(stations[4]);

	// Station control logic and mapping
	// -----------------------------------------------------------------
	station.Control.Enable := TRUE;
	station.Control.Station := ADR(S4);
	station.Control.To := ADR(S5);
	station.Macro.Name := 'S4';
	station.Zone.Name := 'Z4';
	station.Operation.StationQueueControl.ShuttleCapacity := 2;

	// -----------------------------------------------------------------
	CASE station.State OF
		0:
			station.Var.StateInfo := 'Activating station';
			// -----------------------------------------------------------------
			IF station.Control.Active AND station.Control.State = mpTRAFFIC_ST_ON_OPEN THEN
				station.State := station.State + 1;
			END_IF
		1:
			station.Var.StateInfo := 'Create shuttle group';
			// -----------------------------------------------------------------
			station.Commands.Group.Create := TRUE;
			IF station.Group.GroupCreate.Done THEN
				station.Group.ShuttleGroup := station.Group.GroupCreate.ShuttleGroup;
				station.State := 10;
			END_IF;
		10:
			station.Var.StateInfo := 'Create virtual shuttle';
			// -----------------------------------------------------------------
			IF station.Virtual.Shuttle.controlif = 0 THEN
				station.State := station.State + 1;
			ELSE
				station.State := 20;
			END_IF;
		11:
			station.Var.StateInfo := 'Create virtual shuttle';
			// -----------------------------------------------------------------
			station.Commands.CreateVirtualShuttle := TRUE;

			IF station.Virtual.VirtualShCreate.Done THEN
				station.Virtual.Shuttle := station.Virtual.VirtualShCreate.VirtualShuttle;
				station.State := station.State + 1;
			END_IF;
		12:
			station.Var.StateInfo := 'Create virtual shuttle';
			// -----------------------------------------------------------------
			station.Operation.GetShuttleInfo.Shuttle := ADR(station.Virtual.Shuttle);

			station.Commands.GetShuttleInfo := TRUE;

			IF station.Operation.GetShuttleInfo.Done THEN
				station.Virtual.ShuttleID := station.Operation.GetShuttleInfo.ShuttleInfo.ShuttleID;
				station.State := 20;
			END_IF;
		20:
			station.Var.StateInfo := 'Find station zone by name';
			// -----------------------------------------------------------------
			brsmemset(ADR(station.Zone.Zone), 0, SIZEOF(station.Zone.Zone));
			station.Zone.FindZone.Name := station.Zone.Name;
			station.Commands.Zone.Find := TRUE;

			IF station.Zone.FindZone.ZoneFound THEN
				station.Zone.Zone := station.Zone.FindZone.Zone;
				station.State := 30;
			ELSIF station.Zone.FindZone.ZoneNotFound THEN
				station.State := station.State + 1;
			END_IF;
		21:
			station.Var.StateInfo := 'Create zone';
			// -----------------------------------------------------------------
			station.Zone.ZoneCreate.Parameters.BottomLeft.X := 0.000;
			station.Zone.ZoneCreate.Parameters.BottomLeft.Y := 1.440;
			station.Zone.ZoneCreate.Parameters.TopRight.X := 0.240;
			station.Zone.ZoneCreate.Parameters.TopRight.Y := 1.900;
			station.Zone.ZoneCreate.Parameters.Name := station.Zone.Name;
			station.Commands.Zone.Create := TRUE;

			IF station.Zone.ZoneCreate.Done THEN
				// Go back one step and rescan the zones to get the zone reference
				station.State := 20;
			END_IF;
		30:
			station.Var.StateInfo := 'Check if station sequence macro exists';
			// -----------------------------------------------------------------
			IF station.Macro.Shuttle.controlif = 0 THEN
				station.State := station.State + 1;
			ELSE
				station.State := 200;
			END_IF;
		31:
			station.Var.StateInfo := 'Check if station sequence macro exists';
			// -----------------------------------------------------------------
			station.Commands.Macro.Create := TRUE;

			IF station.Macro.MacroCreate.Done THEN
				station.Macro.Shuttle := station.Macro.MacroCreate.MacroShuttle;
				station.State := 200;
			END_IF;

		200:
			// Station sequence
			// ----------------------------------------------------------------------------------------------------------------------------------
			station.Var.StateInfo := 'Initialize station sequence';
			// -----------------------------------------------------------------
			reset_parameters_all;
			station.ShuttleCount := 0;
			brsmemset(ADR(station.Shuttles), 0, SIZEOF(station.Shuttles));
			station.State := station.State + 1;

		201:
			station.Var.StateInfo := 'Waiting for first shuttle to arrive at station';
			// -----------------------------------------------------------------
			IF station.Control.Info.NumOccupyingShuttles > 0 THEN
				station.Shuttles[station.ShuttleCount] := station.Control.Info.LastArrivedShuttle;
				station.ShuttleCount := station.ShuttleCount + 1;
				station.State := station.State + 1;
			END_IF;
		202:
			station.Var.StateInfo := 'Move first shuttle to start position';
			// -----------------------------------------------------------------
			station.Operation.MoveInPlane.Shuttle := ADR(station.Shuttles[0].Shuttle6D);
			station.Operation.MoveInPlane.Parameters.Position.X := 0.120;
			station.Operation.MoveInPlane.Parameters.Position.Y := 1.740;
			station.Operation.MoveInPlane.Parameters.Path :=  mcACP6D_PATH_X_THEN_Y;
			station.Commands.MoveInPlane := TRUE;

			IF station.Operation.MoveInPlane.Done THEN
				station.State := station.State + 1;
			END_IF;
		203:
			station.Var.StateInfo := 'Waiting for second shuttle to arrive at station';
			// -----------------------------------------------------------------
			IF station.Control.Info.NumOccupyingShuttles > 1 THEN
				station.Shuttles[station.ShuttleCount] := station.Control.Info.LastArrivedShuttle;
				station.ShuttleCount := station.ShuttleCount + 1;
				station.State := station.State + 1;
			END_IF;
		204:
			station.Var.StateInfo := 'Move second shuttle to start position';
			// -----------------------------------------------------------------
			station.Operation.MoveInPlane.Shuttle := ADR(station.Shuttles[1].Shuttle6D);
			station.Operation.MoveInPlane.Parameters.Position.X := 0.120;
			station.Operation.MoveInPlane.Parameters.Position.Y := 1.620;
			station.Operation.MoveInPlane.Parameters.Path :=  mcACP6D_PATH_X_THEN_Y;
			station.Commands.MoveInPlane := TRUE;

			IF station.Operation.MoveInPlane.Done THEN
				station.State := 210;
			END_IF;
		210:
			station.Var.StateInfo := 'Init synchronized move';
			// -----------------------------------------------------------------
			reset_parameters_all;
			station.Operation.MoveArc.Parameters.Angular.Angle := 10 * brmTWOPI;

			station.Operation.WaitCommandLabel.TriggerXID := station.Shuttles[0].ShuttleID;
			station.Operation.WaitCommandLabel.TriggerCmdLb := 0;
			station.State := station.State + 1;
		211:
			station.Var.StateInfo := 'Shuttle 1 waits for 0';
			// -----------------------------------------------------------------
			station.Operation.WaitCommandLabel.Shuttle := ADR(station.Shuttles[1].Shuttle6D);
			station.Commands.WaitCommandLabel := TRUE;

			IF station.Operation.WaitCommandLabel.Acknowledge THEN
				station.State := station.State + 1;
			END_IF;
		212:
			station.Var.StateInfo := 'Arc';
			// -----------------------------------------------------------------
			station.Operation.MoveArc.Parameters.Direction := mcACP6D_ARC_CLOCKWISE;
			station.Operation.MoveArc.Parameters.Angular.Center.X := 0;
			station.Operation.MoveArc.Parameters.Angular.Center.Y := -0.060;
			station.Operation.MoveArc.Shuttle := ADR(station.Shuttles[1].Shuttle6D);
			station.Commands.MoveArc := TRUE;

			IF station.Operation.MoveArc.Acknowledge THEN
				station.State := station.State + 1;
			END_IF;
		213:
			station.Var.StateInfo := 'Arc';
			// -----------------------------------------------------------------
			station.Operation.MoveArc.Parameters.Direction := mcACP6D_ARC_CLOCKWISE;
			station.Operation.MoveArc.Parameters.Angular.Center.X := 0;
			station.Operation.MoveArc.Parameters.Angular.Center.Y := 0.060;
			station.Operation.MoveArc.Shuttle := ADR(station.Shuttles[0].Shuttle6D);
			station.Commands.MoveArc := TRUE;

			IF station.Operation.MoveArc.Acknowledge THEN
				station.State := station.State + 1;
			END_IF;
		214:
			station.Var.StateInfo := 'Move to 2nd start pos';
			// -----------------------------------------------------------------
			reset_parameters_all;
			station.Operation.MoveInPlane.Shuttle := ADR(station.Shuttles[0].Shuttle6D);
			station.Operation.MoveInPlane.Parameters.Position.X := 0.180;
			station.Operation.MoveInPlane.Parameters.Position.Y := 1.860;
			station.Commands.MoveInPlane := TRUE;

			IF station.Operation.MoveInPlane.Acknowledge THEN
				station.State := station.State + 1;
			END_IF;
		215:
			station.Var.StateInfo := 'Move to 2nd start pos';
			// -----------------------------------------------------------------
			reset_parameters_all;
			station.Operation.MoveInPlane.Shuttle := ADR(station.Shuttles[1].Shuttle6D);
			station.Operation.MoveInPlane.Parameters.Position.X := 0.060;
			station.Operation.MoveInPlane.Parameters.Position.Y := 1.500;
			station.Commands.MoveInPlane := TRUE;

			IF station.Operation.MoveInPlane.Acknowledge THEN
				station.State := station.State + 1;
			END_IF;
		216:
			station.Var.StateInfo := 'Sync shuttles';
			// -----------------------------------------------------------------
			station.Operation.WaitUntilAllDone.Shuttles[0] := station.Shuttles[0].Shuttle6D;
			station.Operation.WaitUntilAllDone.Shuttles[1] := station.Shuttles[1].Shuttle6D;
			station.Commands.WaitUntilAllDone := TRUE;

			IF station.Operation.WaitUntilAllDone.Done THEN
				station.State := 220;
			END_IF;

		220:
			station.Var.StateInfo := 'Move pattern for slave shuttle';
			// -----------------------------------------------------------------
			reset_parameters_all;
			station.Operation.MoveInPlane.Shuttle := ADR(station.Shuttles[1].Shuttle6D);
			station.Operation.MoveInPlane.Parameters.Mode := mcACP6D_MOVE_RELATIVE;

			station.Operation.WaitCommandLabel.TriggerXID := station.Shuttles[0].ShuttleID;
			station.Operation.WaitCommandLabel.TriggerCmdLb := 0;
			station.State := station.State + 1;
		221:
			station.Var.StateInfo := '';
			// -----------------------------------------------------------------
			station.Operation.WaitCommandLabel.Shuttle := ADR(station.Shuttles[1].Shuttle6D);
			station.Commands.WaitCommandLabel := TRUE;

			IF station.Operation.WaitCommandLabel.Acknowledge THEN
				station.State := station.State + 1;
			END_IF;
		222:
			station.Var.StateInfo := 'Shuttle 1 moves';
			// -----------------------------------------------------------------
			station.Operation.MoveInPlane.Parameters.Position.X := 0.120;
			station.Operation.MoveInPlane.Parameters.Position.Y := 0.0;
			station.Commands.MoveInPlane := TRUE;

			IF station.Operation.MoveInPlane.Acknowledge THEN
				station.State := station.State + 1;
			END_IF;
		223:
			station.Var.StateInfo := 'Shuttle 1 moves';
			// -----------------------------------------------------------------
			station.Operation.MoveInPlane.Parameters.Position.X := 0.000;
			station.Operation.MoveInPlane.Parameters.Position.Y := 0.120;
			station.Commands.MoveInPlane := TRUE;

			IF station.Operation.MoveInPlane.Acknowledge THEN
				station.State := station.State + 1;
			END_IF;
		224:
			station.Var.StateInfo := 'Shuttle 1 moves';
			// -----------------------------------------------------------------
			station.Operation.MoveInPlane.Parameters.Position.X := -0.120;
			station.Operation.MoveInPlane.Parameters.Position.Y := 0.0;
			station.Commands.MoveInPlane := TRUE;

			IF station.Operation.MoveInPlane.Acknowledge THEN
				station.State := station.State + 1;
			END_IF;
		225:
			station.Var.StateInfo := 'Shuttle 1 moves';
			// -----------------------------------------------------------------
			station.Operation.MoveInPlane.Parameters.Position.X := 0.000;
			station.Operation.MoveInPlane.Parameters.Position.Y := 0.120;
			station.Commands.MoveInPlane := TRUE;

			IF station.Operation.MoveInPlane.Acknowledge THEN
				station.State := station.State + 1;
			END_IF;
		226:
			station.Var.StateInfo := 'Shuttle 1 moves';
			// -----------------------------------------------------------------
			station.Operation.MoveInPlane.Parameters.Position.X := 0.120;
			station.Operation.MoveInPlane.Parameters.Position.Y := 0.0;
			station.Commands.MoveInPlane := TRUE;

			IF station.Operation.MoveInPlane.Acknowledge THEN
				station.State := station.State + 1;
			END_IF;
		227:
			station.Var.StateInfo := 'Shuttle 1 moves';
			// -----------------------------------------------------------------
			station.Operation.MoveInPlane.Parameters.Position.X := 0.000;
			station.Operation.MoveInPlane.Parameters.Position.Y := 0.120;
			station.Commands.MoveInPlane := TRUE;

			IF station.Operation.MoveInPlane.Acknowledge THEN
				station.State := station.State + 1;
			END_IF;
		228:
			station.Var.StateInfo := 'Shuttle 1 moves';
			// -----------------------------------------------------------------
			station.Operation.MoveInPlane.Parameters.Position.X := -0.120;
			station.Operation.MoveInPlane.Parameters.Position.Y := 0.0;
			station.Commands.MoveInPlane := TRUE;

			IF station.Operation.MoveInPlane.Acknowledge THEN
				station.State := 240;
			END_IF;

		240:
			station.Var.StateInfo := 'Move pattern for master shuttle';
			// -----------------------------------------------------------------
			reset_parameters_all;
			station.Operation.MoveInPlane.Shuttle := ADR(station.Shuttles[0].Shuttle6D);
			station.Operation.MoveInPlane.Parameters.Mode := mcACP6D_MOVE_RELATIVE;
			station.State := station.State + 1;
		241:
			station.Var.StateInfo := 'Shuttle 0 moves';
			// -----------------------------------------------------------------
			station.Operation.MoveInPlane.Parameters.Position.X := -0.120;
			station.Operation.MoveInPlane.Parameters.Position.Y := 0.0;
			station.Commands.MoveInPlane := TRUE;

			IF station.Operation.MoveInPlane.Acknowledge THEN
				station.State := station.State + 1;
			END_IF;
		242:
			station.Var.StateInfo := 'Shuttle 0 moves';
			// -----------------------------------------------------------------
			station.Operation.MoveInPlane.Parameters.Position.X := 0.000;
			station.Operation.MoveInPlane.Parameters.Position.Y := -0.120;
			station.Commands.MoveInPlane := TRUE;

			IF station.Operation.MoveInPlane.Acknowledge THEN
				station.State := station.State + 1;
			END_IF;
		243:
			station.Var.StateInfo := 'Shuttle 0 moves';
			// -----------------------------------------------------------------
			station.Operation.MoveInPlane.Parameters.Position.X := 0.120;
			station.Operation.MoveInPlane.Parameters.Position.Y := 0.0;
			station.Commands.MoveInPlane := TRUE;

			IF station.Operation.MoveInPlane.Acknowledge THEN
				station.State := station.State + 1;
			END_IF;
		244:
			station.Var.StateInfo := 'Shuttle 0 moves';
			// -----------------------------------------------------------------
			station.Operation.MoveInPlane.Parameters.Position.X := 0.000;
			station.Operation.MoveInPlane.Parameters.Position.Y := -0.120;
			station.Commands.MoveInPlane := TRUE;

			IF station.Operation.MoveInPlane.Acknowledge THEN
				station.State := station.State + 1;
			END_IF;
		245:
			station.Var.StateInfo := 'Shuttle 0 moves';
			// -----------------------------------------------------------------
			station.Operation.MoveInPlane.Parameters.Position.X := -0.120;
			station.Operation.MoveInPlane.Parameters.Position.Y := 0.0;
			station.Commands.MoveInPlane := TRUE;

			IF station.Operation.MoveInPlane.Acknowledge THEN
				station.State := station.State + 1;
			END_IF;
		246:
			station.Var.StateInfo := 'Shuttle 0 moves';
			// -----------------------------------------------------------------
			station.Operation.MoveInPlane.Parameters.Position.X := 0.000;
			station.Operation.MoveInPlane.Parameters.Position.Y := -0.120;
			station.Commands.MoveInPlane := TRUE;

			IF station.Operation.MoveInPlane.Acknowledge THEN
				station.State := station.State + 1;
			END_IF;
		247:
			station.Var.StateInfo := 'Shuttle 0 moves';
			// -----------------------------------------------------------------
			station.Operation.MoveInPlane.Parameters.Position.X := 0.120;
			station.Operation.MoveInPlane.Parameters.Position.Y := 0.0;
			station.Commands.MoveInPlane := TRUE;

			IF station.Operation.MoveInPlane.Acknowledge THEN
				station.State := 1000;
			END_IF;

		1000:
			station.Var.StateInfo := 'Sync shuttles';
			// -----------------------------------------------------------------
			station.Operation.WaitUntilAllDone.Shuttles[0] := station.Shuttles[0].Shuttle6D;
			station.Operation.WaitUntilAllDone.Shuttles[1] := station.Shuttles[1].Shuttle6D;
			station.Commands.WaitUntilAllDone := TRUE;

			IF station.Operation.WaitUntilAllDone.Done THEN
				station.State := station.State + 1;
			END_IF;
		1001:
			station.Var.StateInfo := 'Clear group';
			// -----------------------------------------------------------------
			station.Commands.Group.Clear := TRUE;

			IF station.Group.GroupClear.Done THEN
				station.State := station.State + 1;
			END_IF;
		1002:
			// Return shuttles to the traffic network
			// ----------------------------------------------------------------------------------------------------------------------------------
			station.Var.StateInfo := 'Move shuttles to exit positions';
			// -----------------------------------------------------------------
			reset_parameters_all;

			station.Operation.MoveInPlane.Shuttle := ADR(station.Shuttles[0].Shuttle6D);
			station.Operation.MoveInPlane.Parameters.Path := mcACP6D_PATH_X_THEN_Y;
			station.Operation.MoveInPlane.Parameters.Position.X := 0.180;
			station.Operation.MoveInPlane.Parameters.Position.Y := 1.860;
			station.Commands.MoveInPlane := TRUE;

			IF station.Operation.MoveInPlane.Done THEN
				station.State := station.State + 1;
			END_IF;
		1003:
			station.Var.StateInfo := 'Move shuttles to exit positions';
			// -----------------------------------------------------------------
			station.Operation.MoveInPlane.Shuttle := ADR(station.Shuttles[1].Shuttle6D);
			station.Operation.MoveInPlane.Parameters.Path := mcACP6D_PATH_X_THEN_Y;
			station.Operation.MoveInPlane.Parameters.Position.X := 0.060;
			station.Operation.MoveInPlane.Parameters.Position.Y := 1.860;
			station.Commands.MoveInPlane := TRUE;

			IF station.Operation.MoveInPlane.Done THEN
				station.State := station.State + 1;
			END_IF;
		1004:
			station.Var.StateInfo := 'Release shuttles';
			// -----------------------------------------------------------------
			station.Operation.StationQueueControl.ShuttleList[0] := station.Shuttles[0];
			station.Operation.StationQueueControl.ShuttleList[1] := station.Shuttles[1];
			station.Commands.Release := TRUE;

			IF station.Operation.StationQueueControl.ShuttleReleaseDone THEN
				station.State := station.State + 1;
			END_IF;
		1005:
			station.Var.StateInfo := 'Wait until shuttles at the station have all left';
			// -----------------------------------------------------------------
			station.Commands.Zone.GetBarrierInfo := TRUE;

			IF station.Zone.ZoneGetBarrierInfo.Done THEN
				station.Commands.Zone.GetBarrierInfo := FALSE;
				IF station.Zone.ZoneGetBarrierInfo.BarrierInfo.NumberOfShuttles = 0 THEN
					station.State := 200;
				END_IF;
			END_IF;
	END_CASE;

	// Reset station commands when state changes
	IF station.State <> station.Var.PreviousState THEN
		station.Var.PreviousState := station.State;
		brsmemset(ADR(station.Commands), 0, SIZEOF(station.Commands));
	END_IF;

END_ACTION
```
